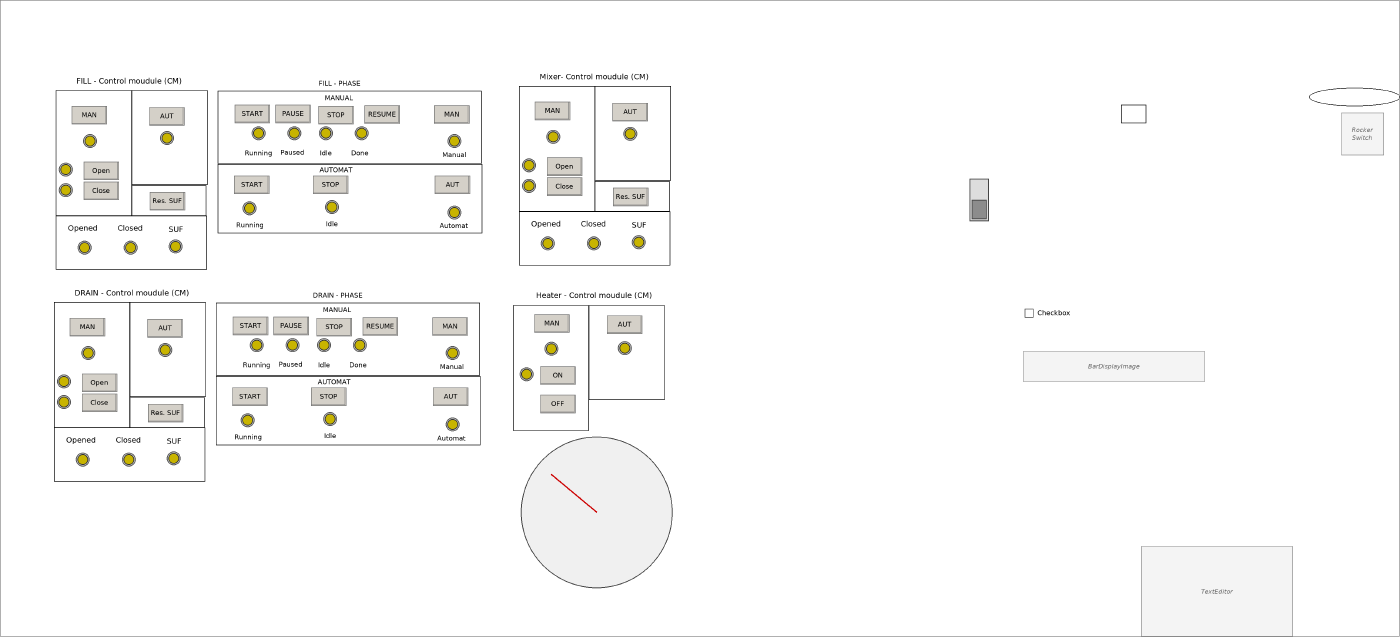
VISUALIZATION Visualization  // 2309x1052
    Rectangle (217,149 125x156)
    Rectangle (217,306 123x50)
    Rectangle (92,149 125x207)
    Rectangle (359,271 436x114)
    Rectangle (92,356 249x89)
    Checkbox (1688,502 150x30), "Checkbox"
    BarDisplayImage (1687,580 300x50), style: BarDisplayImage-Gray, scale format: %.1f, scale 0..100
    DipSwitch (1580,295 70x70), behaviour: TOGGLE, style: Switch-DipSwitch-Gray
    RockerSwitch (2212,186 70x70), behaviour: TOGGLE, style: Switch-RockerSwitch-Gray
    TextEditor (1882,902 250x150)
        p4127561890: Courier New
    Ellipse (2159,145 150x30)
    Rectangle (1849,173 41x30)
    Button (246,177 58x30), "AUT"
        OnMouseClick: toggle Global.Tank1.ValveFilling.Cmd.AutCtrl
    Button (118,175 58x30), "MAN"
        OnMouseClick: toggle Global.Tank1.ValveFilling.Cmd.ManCtrl
    Label (123,125 212x18), "FILL - Control moudule (CM)"
    Button (138,267 58x30), "Open"
        OnMouseClick: toggle Global.Tank1.ValveFilling.Cmd.OpenMan
    Button (138,300 58x30), "Close"
        OnMouseClick: toggle Global.Tank1.ValveFilling.Cmd.CloseMan
    Lamp1 (262,215 27x26), variable: Global.Tank1.ValveFilling.State.AutCtrl, style: Lamp-Lamp1-Yellow
    Lamp1 (135,220 27x26), variable: Global.Tank1.ValveFilling.State.ManCtrl, style: Lamp-Lamp1-Yellow
    Lamp1 (126,396 27x26), variable: Global.Tank1.ValveFilling.State.Open, style: Lamp-Lamp1-Yellow
    Lamp1 (202,396 27x26), variable: Global.Tank1.ValveFilling.State.Closed, style: Lamp-Lamp1-Yellow
    Lamp1 (276,394 27x26), variable: Global.Tank1.ValveFilling.State.StartupFail, style: Lamp-Lamp1-Yellow
    Button (247,317 58x30), "Res. SUF"
        OnMouseClick: toggle Global.Tank1.ValveFilling.Cmd.ResetSUF
    Label (109,368 53x18), "Opened"
    Label (191,368 53x18), "Closed"
    Label (275,370 33x18), "SUF"
    Lamp1 (95,267 27x26), variable: Global.Tank1.ValveFilling.State.OpenOut, style: Lamp-Lamp1-Yellow
    Lamp1 (95,301 27x26), variable: Global.Tank1.ValveFilling.State.CloseOut, style: Lamp-Lamp1-Yellow
    Rectangle (359,150 435x120)
    Lamp1 (413,207 27x26), variable: Main_Batch.FB_Tank_1.FillingPhase.FillingPhase.State.Running, style: Lamp-Lamp1-Yellow
    Lamp1 (472,207 27x26), variable: Global.Tank1.Filling.State.Paused, style: Lamp-Lamp1-Yellow
    Lamp1 (524,207 27x26), variable: Global.Tank1.Filling.State.Idle, style: Lamp-Lamp1-Yellow
    Lamp1 (583,207 27x26), variable: Global.Tank1.Filling.State.Done, style: Lamp-Lamp1-Yellow
    Label (485,123 150x30), "FILL - PHASE"
    Label (400,238 53x30), "Running"
    Label (456,237 53x30), "Paused"
    Label (511,238 53x30), "Idle"
    Label (567,238 53x30), "Done"
    Button (717,290 58x30), "AUT"
        OnMouseClick: toggle Global.Tank1.Filling.Cmd.AutCtrl
    Button (716,174 58x30), "MAN"
        OnMouseClick: toggle Global.Tank1.Filling.Cmd.ManCtrl
    Lamp1 (736,338 27x26), variable: Global.Tank1.Filling.State.AutCtrl, style: Lamp-Lamp1-Yellow
    Lamp1 (736,220 27x26), variable: Global.Tank1.Filling.State.ManCtrl, style: Lamp-Lamp1-Yellow
    Button (387,173 58x30), "START"
        OnMouseClick: toggle Global.Tank1.Filling.Cmd.StartMan
    Button (454,173 58x30), "PAUSE"
        OnMouseClick: toggle Global.Tank1.Filling.Cmd.PauseMan
    Button (525,175 58x30), "STOP"
        OnMouseClick: toggle Global.Tank1.Filling.Cmd.StopMan
    Button (601,174 58x30), "RESUME"
        OnMouseClick: toggle Global.Tank1.Filling.Cmd.ResumeMan
    Button (386,290 58x30), "START"
        OnMouseClick: toggle Global.Tank1.Filling.Cmd.StartAut
    Button (516,290 58x30), "STOP"
        OnMouseClick: toggle Global.Tank1.Filling.Cmd.StopAut
    Lamp1 (398,331 27x26), variable: Global.Tank1.Filling.State.Running, style: Lamp-Lamp1-Yellow
    Lamp1 (534,329 27x26), variable: Global.Tank1.Filling.State.Idle, style: Lamp-Lamp1-Yellow
    Label (484,147 150x30), "MANUAL"
    Label (479,266 150x30), "AUTOMAT"
    Label (386,357 53x30), "Running"
    Label (521,355 53x30), "Idle"
    Rectangle (214,499 125x156)
    Rectangle (214,656 123x50)
    Rectangle (89,499 125x207)
    Rectangle (356,621 436x114)
    Rectangle (89,706 249x89)
    Button (243,527 58x30), "AUT"
        OnMouseClick: toggle Global.Tank1.ValveDraining.Cmd.AutCtrl
    Button (115,525 58x30), "MAN"
        OnMouseClick: toggle Global.Tank1.ValveDraining.Cmd.ManCtrl
    Label (120,475 212x18), "DRAIN - Control moudule (CM)"
    Button (135,617 58x30), "Open"
        OnMouseClick: toggle Global.Tank1.ValveDraining.Cmd.OpenMan
    Button (135,650 58x30), "Close"
        OnMouseClick: toggle Global.Tank1.ValveDraining.Cmd.CloseMan
    Lamp1 (259,565 27x26), variable: Global.Tank1.ValveDraining.State.AutCtrl, style: Lamp-Lamp1-Yellow
    Lamp1 (132,570 27x26), variable: Global.Tank1.ValveDraining.State.ManCtrl, style: Lamp-Lamp1-Yellow
    Lamp1 (123,746 27x26), variable: Global.Tank1.ValveFilling.State.Open, style: Lamp-Lamp1-Yellow
    Lamp1 (199,746 27x26), variable: Global.Tank1.ValveFilling.State.Closed, style: Lamp-Lamp1-Yellow
    Lamp1 (273,744 27x26), variable: Global.Tank1.ValveDraining.State.StartupFail, style: Lamp-Lamp1-Yellow
    Button (244,667 58x30), "Res. SUF"
        OnMouseClick: toggle Global.Tank1.ValveDraining.Cmd.ResetSUF
    Label (106,718 53x18), "Opened"
    Label (188,718 53x18), "Closed"
    Label (272,720 33x18), "SUF"
    Lamp1 (92,617 27x26), variable: Global.Tank1.ValveDraining.State.OpenOut, style: Lamp-Lamp1-Yellow
    Lamp1 (92,651 27x26), variable: Global.Tank1.ValveDraining.State.CloseOut, style: Lamp-Lamp1-Yellow
    Rectangle (356,500 435x120)
    Lamp1 (410,557 27x26), variable: Global.Tank1.Draining.State.Running, style: Lamp-Lamp1-Yellow
    Lamp1 (469,557 27x26), variable: Global.Tank1.Draining.State.Paused, style: Lamp-Lamp1-Yellow
    Lamp1 (521,557 27x26), variable: Global.Tank1.Draining.State.Idle, style: Lamp-Lamp1-Yellow
    Lamp1 (580,557 27x26), variable: Global.Tank1.Draining.State.Done, style: Lamp-Lamp1-Yellow
    Label (482,473 150x30), "DRAIN - PHASE"
    Label (397,588 53x30), "Running"
    Label (453,587 53x30), "Paused"
    Label (508,588 53x30), "Idle"
    Label (564,588 53x30), "Done"
    Button (714,640 58x30), "AUT"
        OnMouseClick: toggle Global.Tank1.Draining.Cmd.AutCtrl
    Button (713,524 58x30), "MAN"
        OnMouseClick: toggle Global.Tank1.Draining.Cmd.ManCtrl
    Lamp1 (733,688 27x26), variable: Global.Tank1.Draining.State.AutCtrl, style: Lamp-Lamp1-Yellow
    Lamp1 (733,570 27x26), variable: Global.Tank1.Draining.State.ManCtrl, style: Lamp-Lamp1-Yellow
    Button (384,523 58x30), "START"
        OnMouseClick: toggle Global.Tank1.Draining.Cmd.StartMan
    Button (451,523 58x30), "PAUSE"
        OnMouseClick: toggle Global.Tank1.Draining.Cmd.PauseMan
    Button (522,525 58x30), "STOP"
        OnMouseClick: toggle Global.Tank1.Draining.Cmd.StopMan
    Button (598,524 58x30), "RESUME"
        OnMouseClick: toggle Global.Tank1.Draining.Cmd.ResumeMan
    Button (383,640 58x30), "START"
        OnMouseClick: toggle Global.Tank1.Draining.Cmd.StartAut
    Button (513,640 58x30), "STOP"
        OnMouseClick: toggle Global.Tank1.Draining.Cmd.StopAut
    Lamp1 (395,681 27x26), variable: Global.Tank1.Draining.State.Running, style: Lamp-Lamp1-Yellow
    Lamp1 (531,679 27x26), variable: Global.Tank1.Draining.State.Idle, style: Lamp-Lamp1-Yellow
    Label (481,497 150x30), "MANUAL"
    Label (476,616 150x30), "AUTOMAT"
    Label (383,707 53x30), "Running"
    Label (518,705 53x30), "Idle"
    Label (723,241 53x30), "Manual"
    Label (719,591 53x30), "Manual"
    Label (722,358 53x30), "Automat"
    Label (718,709 53x30), "Automat"
    Rectangle (981,142 125x156)
    Rectangle (981,299 123x50)
    Rectangle (856,142 125x207)
    Rectangle (856,349 249x89)
    Button (1010,170 58x30), "AUT"
        OnMouseClick: toggle Global.Tank1.Mixer.Cmd.AutCtrl
    Button (882,168 58x30), "MAN"
        OnMouseClick: toggle Global.Tank1.Mixer.Cmd.ManCtrl
    Label (887,118 212x18), "Mixer- Control moudule (CM)"
    Button (902,260 58x30), "Open"
        OnMouseClick: toggle Global.Tank1.ValveFilling.Cmd.OpenMan
    Button (902,293 58x30), "Close"
        OnMouseClick: toggle Global.Tank1.ValveFilling.Cmd.CloseMan
    Lamp1 (1026,208 27x26), variable: Global.Tank1.Mixer.State.AutCtrl, style: Lamp-Lamp1-Yellow
    Lamp1 (899,213 27x26), variable: Global.Tank1.Mixer.State.ManCtrl, style: Lamp-Lamp1-Yellow
    Lamp1 (890,389 27x26), variable: Global.Tank1.ValveFilling.State.Open, style: Lamp-Lamp1-Yellow
    Lamp1 (966,389 27x26), variable: Global.Tank1.ValveFilling.State.Closed, style: Lamp-Lamp1-Yellow
    Lamp1 (1040,387 27x26), variable: Global.Tank1.ValveFilling.State.StartupFail, style: Lamp-Lamp1-Yellow
    Button (1011,310 58x30), "Res. SUF"
        OnMouseClick: toggle Global.Tank1.ValveFilling.Cmd.ResetSUF
    Label (873,361 53x18), "Opened"
    Label (955,361 53x18), "Closed"
    Label (1039,363 33x18), "SUF"
    Lamp1 (859,260 27x26), variable: Global.Tank1.ValveFilling.State.OpenOut, style: Lamp-Lamp1-Yellow
    Lamp1 (859,294 27x26), variable: Global.Tank1.ValveFilling.State.CloseOut, style: Lamp-Lamp1-Yellow
    Label (881,479 212x18), "Heater - Control moudule (CM)"
    Rectangle (846,504 125x207)
    Rectangle (971,504 125x156)
    Button (881,519 58x30), "MAN"
        OnMouseClick: toggle Global.Tank1.Heater.Cmd.ManCtrl
    Button (1001,521 58x30), "AUT"
        OnMouseClick: toggle Global.Tank1.Heater.Cmd.AutCtrl
    Lamp1 (896,563 27x26), variable: Global.Tank1.Heater.State.ManCtrl, style: Lamp-Lamp1-Yellow
    Lamp1 (1017,562 27x26), variable: Global.Tank1.Heater.State.AutCtrl, style: Lamp-Lamp1-Yellow
    Button (891,605 58x30), "ON"
        OnMouseClick: toggle Global.Tank1.Heater.Cmd.TurnOnMan
    Button (891,652 58x30), "OFF"
        OnMouseClick: toggle Global.Tank1.Heater.Cmd.TurnOffMan
    Lamp1 (855,605 27x26), variable: Global.Tank1.Heater.State.EnableOut, style: Lamp-Lamp1-Yellow
    Meter360 (859,721 250x250), value: Global.Tank1.Heater.State.HeatingOut, style: Meter-Meter360-Gray, scale format: %.1f, scale 0..100
END_VISUALIZATION

(* stored: Version 1.1.0.1, ProductVersion 3.1.4024.15
   Visu Visualization: Id {a6343251-0068-49ba-9adb-31cb88a6e465} *)
